# EPICS autosave request: softGlueApp/Db/IF_tracker_settings.req
$(P)$(H)IF_tracker-$(N)_CLOCK_Signal
$(P)$(H)IF_tracker-$(N)_EN_Signal
$(P)$(H)IF_tracker-$(N)_CLEAR_Signal
$(P)$(H)IF_tracker-$(N)_MISSCLR_Signal
$(P)$(H)IF_tracker-$(N)_LOAD_Signal
$(P)$(H)IF_tracker-$(N)_LDVAL
$(P)$(H)IF_tracker-$(N)_MISS_Signal
